{attribute 'GeneratedUsingTerminal: KL3041'}
{attribute addProperty BoxType "KL3041"}
{attribute addProperty Id "Channel_1AT %Q*Channel_6576A6810"}
{attribute addProperty CRC "1632160004"}
{attribute addProperty Size "0"}
TYPE KL3041_6148C904 :
STRUCT
	{attribute addProperty Name "Channel_1"}
	Channel_1 : Channel_6576A681;
END_STRUCT
END_TYPE

(* stored: Version 1.2.0.0, ProductVersion 3.1.4024.9
   DUT KL3041_6148C904: Id {8bffe8b4-a9f6-4fa9-aa9a-0ca38df5ae94} *)
